{attribute 'qualified_only'}
{attribute 'strict'}
TYPE E_Actuator :
(
	eDisabled					:= 0,					// Stan nieaktywnosci             	
	eAborted                    := 1,                   // Stan bezpiecznego zatrzymania  
	eAborting                   := 2,                   // Stan bezpiecznego zatrzymywania
	eError                      := 3,                   // Stan bledu 				                                
	ePreparingToReady           := 7,                   // Stan przygotowywania do gotowosci           
	ePreparingToDisable         := 8,                   // Stan przygotowywania do nieaktywnosci                               
	eReady                      := 10,					// Stan gotowosci
	eResetting					:= 13,					// Stan resetowania bledu
	eRunningToPosition1			:= 15,       
	eRunningToPosition2			:= 16,                                          
	eRunning					:= 98,	                // Stan wykonywania ruchu 
    eNotdone                    := 99,	                // Stan niezakonczenia wykonywanego	                                     
    eDone                       := 100,                  // Stan zakonczenia wykonywanego ruchu   
	eDoneToPosition1            := 101,                  // Stan zakonczenia wykonywanego ruchu 
	eDoneToPosition2            := 102                  // Stan zakonczenia wykonywanego ruchu  
);
END_TYPE

(* stored: Version 1.1.0.1, ProductVersion 3.1.4026.13, FileIdentifier 0d73ab8af575d09c659d33693da8a57723c4bf68, FileSignature 7bcccd7b0b2a4e949f7cbbbb7d0aaefa847353d24a04861aa35ac6c759b9af05c1dd42af95f6e33696a6bdc6e634bab6041307e0a6cc384bbcbc9a5dbe2d7ef7ffc5f512a21e6c1f00d4ca7d112f1b258323cafcf6658d1be7476c07e83bcfe046a2f791a9945d078fa049bd4a720f7dbb435e62f5cf1ad3f58268f878814a3bcef1d2b975798408f4d8502f5455aac1d5b924c2de93ecfdf6419cb949269ff192394ecab7785193c0e09df442c6c6aee8badbcf302a82c183cc498a79bd08c79f8491ea8910fe20c50f2644ce9c38957f4041d2bcf18a4582f982fe9b62f83543873898b17786b7e6540e1ec229e6d31c7971a4e84c71d4159f7c8ffce6ce63
   DUT E_Actuator: Id {5e892cf6-3ebb-48e8-a388-0f04bd49a3db} *)
